PROGRAM POU_1
VAR
END_VAR

END_PROGRAM

(* stored: Version 1.1.0.1, ProductVersion 3.1.4024.12
   POU POU_1: Id {760c808e-3274-4efc-b5cc-060550d4033a}, SpecialFunc None *)
